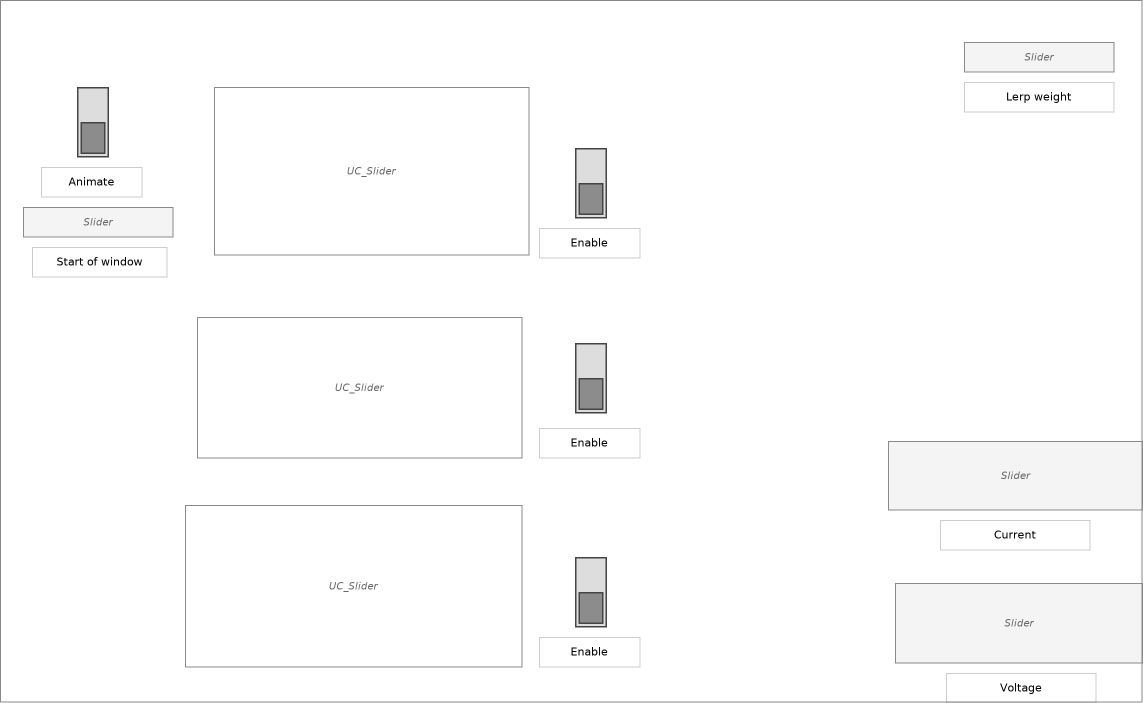
VISUALIZATION Visualization  // 1143x703
    Frame (214,87 315x168)
        shows UC_Slider(PT := MAIN.BackgroundRate.PT, Start := 1, End := 150, Label := 'Background')
    Frame (197,317 325x141)
        shows UC_Slider(PT := MAIN.WhiteRate.PT, Start := 1, End := 75, Label := 'White')
    Frame (185,505 337x162)
        shows UC_Slider(PT := MAIN.ShortredRate.PT, Start := 1, End := 75, Label := 'Shorted')
    DipSwitch (556,148 70x70), variable: MAIN.AddBackground, behaviour: TOGGLE, style: Switch-DipSwitch-Gray
    DipSwitch (556,557 70x70), variable: MAIN.AddShortedLayer, behaviour: TOGGLE, style: Switch-DipSwitch-Gray
    DipSwitch (556,343 70x70), variable: MAIN.AddWhiteLayer, behaviour: TOGGLE, style: Switch-DipSwitch-Gray
    DipSwitch (58,87 70x70), variable: MAIN.AnimateBackgroud, behaviour: TOGGLE, style: Switch-DipSwitch-Gray
    Slider (964,42 150x30), variable: MAIN.weight, scale 0..1
    Textfield (964,82 150x30), "Lerp weight"
    Textfield (41,167 101x30), "Animate"
    Slider (888,441 255x69), variable: MAIN.WhiteRate.PT, scale 1..75
    Slider (895,583 248x80), variable: MAIN.weight, scale 0..1
    Textfield (940,520 150x30), "Current"
    Textfield (946,673 150x30), "Voltage"
    Slider (23,207 150x30), variable: MAIN.backgroundOffset, scale 0..1000
    Textfield (539,228 101x30), "Enable"
    Textfield (539,428 101x30), "Enable"
    Textfield (539,637 101x30), "Enable"
    Textfield (32,247 135x30), "Start of window"
END_VISUALIZATION

(* stored: Version 1.1.0.1
   Visu Visualization: Id {4265dd05-045e-44c3-9202-7c2fa09d9c1a} *)
